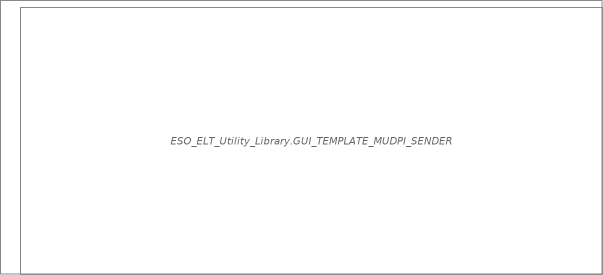
VISUALIZATION GUI_MUDPI_SENDER  // 603x275
    Frame (20,7 583x268)
        shows ESO_ELT_Utility_Library.GUI_TEMPLATE_MUDPI_SENDER(m_Instance := MAIN2.fbSender)
END_VISUALIZATION

(* stored: Version 1.1.0.1, ProductVersion 3.1.4024.11
   Visu GUI_MUDPI_SENDER: Id {efff83ac-22c4-4fc0-85fc-b3f98d8ba69a} *)
